SYSTEM washer_detector
  (* Version 1.0, 2024-11-25, obotnar *)
  APPLICATION washer_detectorApp
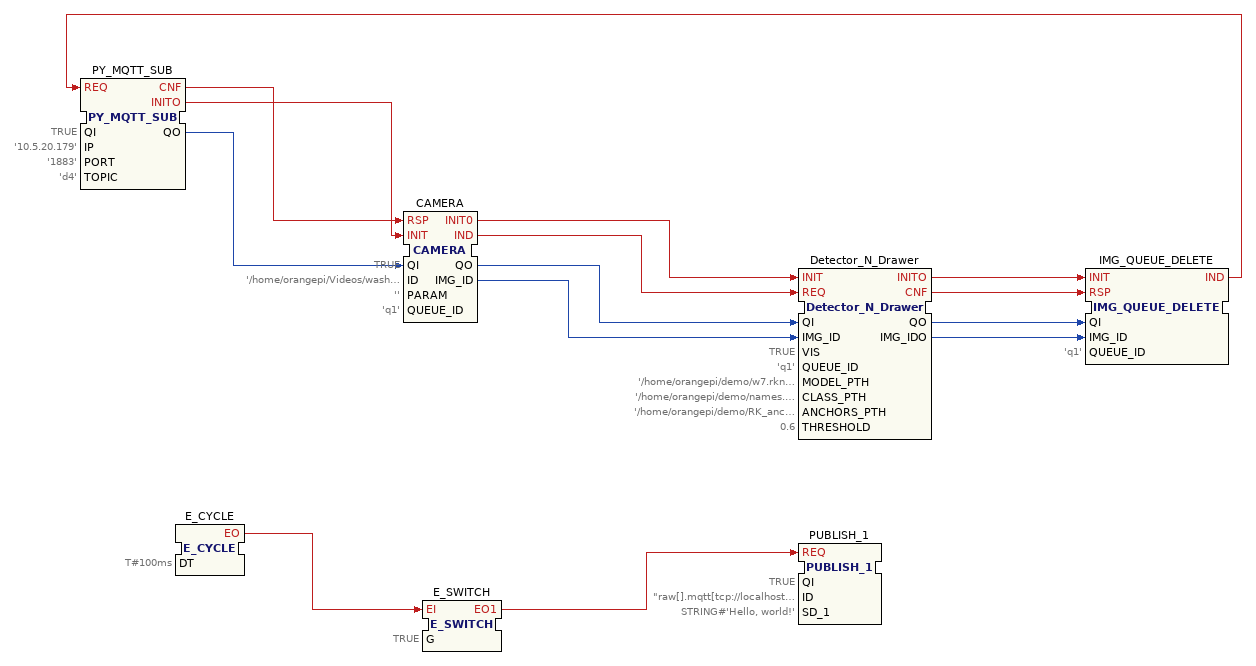
    FBS
      CAMERA : CAMERA(QI := TRUE, ID := '/home/orangepi/Videos/washer.webm', PARAM := '', QUEUE_ID := 'q1');
      IMG_QUEUE_DELETE : IMG_QUEUE_DELETE(QUEUE_ID := 'q1');
      Detector_N_Drawer : Detector_N_Drawer(VIS := TRUE, QUEUE_ID := 'q1', MODEL_PTH := '/home/orangepi/demo/w7.rknn', CLASS_PTH := '/home/orangepi/demo/names.txt', ANCHORS_PTH := '/home/orangepi/demo/RK_anchors.txt', THRESHOLD := 0.6);
      PY_MQTT_SUB : PY_MQTT_SUB(QI := TRUE, IP := '10.5.20.179', PORT := '1883', TOPIC := 'd4');
      E_SWITCH : E_SWITCH(G := TRUE);
      PUBLISH_1 : PUBLISH_1(QI := TRUE, ID := "raw[].mqtt[tcp://localhost:1883, forte, d4]", SD_1 := STRING#'Hello, world!');
      E_CYCLE : E_CYCLE(DT := T#100ms);
    END_FBS
    EVENT_CONNECTIONS
      CAMERA.INIT0 TO Detector_N_Drawer.INIT;
      CAMERA.IND TO Detector_N_Drawer.REQ;
      Detector_N_Drawer.INITO TO IMG_QUEUE_DELETE.INIT;
      Detector_N_Drawer.CNF TO IMG_QUEUE_DELETE.RSP;
      PY_MQTT_SUB.CNF TO CAMERA.RSP;
      PY_MQTT_SUB.INITO TO CAMERA.INIT;
      IMG_QUEUE_DELETE.IND TO PY_MQTT_SUB.REQ;
      E_SWITCH.EO1 TO PUBLISH_1.REQ;
      E_CYCLE.EO TO E_SWITCH.EI;
    END_CONNECTIONS
    DATA_CONNECTIONS
      Detector_N_Drawer.QO TO IMG_QUEUE_DELETE.QI;
      Detector_N_Drawer.IMG_IDO TO IMG_QUEUE_DELETE.IMG_ID;
      CAMERA.QO TO Detector_N_Drawer.QI;
      CAMERA.IMG_ID TO Detector_N_Drawer.IMG_ID;
      PY_MQTT_SUB.QO TO CAMERA.QI;
    END_CONNECTIONS
  END_APPLICATION
  DEVICE FORTE_PC : FORTE_PC(MGR_ID := "10.5.20.198:62499" (* Device manager socket ID *))
    {SET_ATTRIBUTE(Profile, HOLOBLOC)}
    RESOURCE EMB_RES : EMB_RES
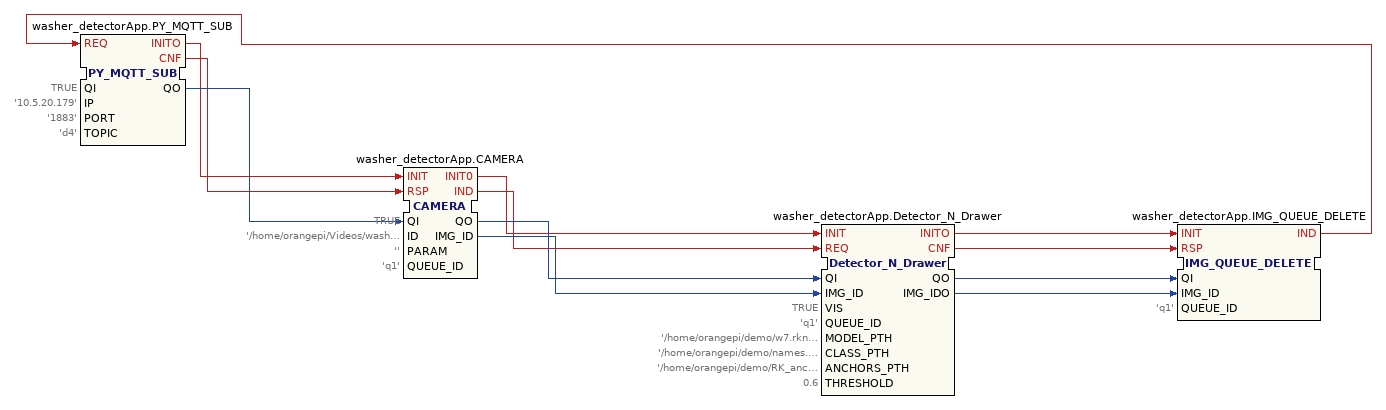
      FBS
        washer_detectorApp.PY_MQTT_SUB : PY_MQTT_SUB(QI := TRUE, IP := '10.5.20.179', PORT := '1883', TOPIC := 'd4');
        washer_detectorApp.CAMERA : CAMERA(QI := TRUE, ID := '/home/orangepi/Videos/washer.webm', PARAM := '', QUEUE_ID := 'q1');
        washer_detectorApp.Detector_N_Drawer : Detector_N_Drawer(VIS := TRUE, QUEUE_ID := 'q1', MODEL_PTH := '/home/orangepi/demo/w7.rknn', CLASS_PTH := '/home/orangepi/demo/names.txt', ANCHORS_PTH := '/home/orangepi/demo/RK_anchors.txt', THRESHOLD := 0.6);
        washer_detectorApp.IMG_QUEUE_DELETE : IMG_QUEUE_DELETE(QUEUE_ID := 'q1');
      END_FBS
      EVENT_CONNECTIONS
        washer_detectorApp.PY_MQTT_SUB.INITO TO washer_detectorApp.CAMERA.INIT;
        washer_detectorApp.PY_MQTT_SUB.CNF TO washer_detectorApp.CAMERA.RSP;
        washer_detectorApp.CAMERA.INIT0 TO washer_detectorApp.Detector_N_Drawer.INIT;
        washer_detectorApp.CAMERA.IND TO washer_detectorApp.Detector_N_Drawer.REQ;
        washer_detectorApp.Detector_N_Drawer.INITO TO washer_detectorApp.IMG_QUEUE_DELETE.INIT;
        washer_detectorApp.Detector_N_Drawer.CNF TO washer_detectorApp.IMG_QUEUE_DELETE.RSP;
        washer_detectorApp.IMG_QUEUE_DELETE.IND TO washer_detectorApp.PY_MQTT_SUB.REQ;
      END_CONNECTIONS
      DATA_CONNECTIONS
        washer_detectorApp.PY_MQTT_SUB.QO TO washer_detectorApp.CAMERA.QI;
        washer_detectorApp.CAMERA.QO TO washer_detectorApp.Detector_N_Drawer.QI;
        washer_detectorApp.CAMERA.IMG_ID TO washer_detectorApp.Detector_N_Drawer.IMG_ID;
        washer_detectorApp.Detector_N_Drawer.QO TO washer_detectorApp.IMG_QUEUE_DELETE.QI;
        washer_detectorApp.Detector_N_Drawer.IMG_IDO TO washer_detectorApp.IMG_QUEUE_DELETE.IMG_ID;
      END_CONNECTIONS
    END_RESOURCE
  END_DEVICE
  DEVICE FORTE_PC_1 : FORTE_PC(MGR_ID := "localhost:61499" (* Device manager socket ID *))
    {SET_ATTRIBUTE(Profile, HOLOBLOC)}
    RESOURCE EMB_RES : EMB_RES
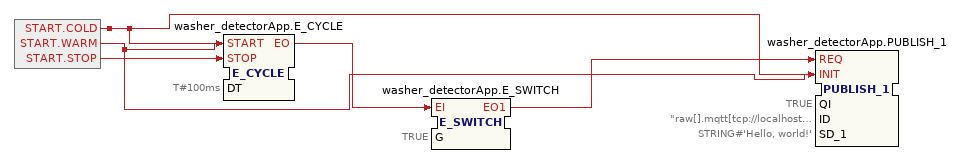
      FBS
        washer_detectorApp.PUBLISH_1 : PUBLISH_1(QI := TRUE, ID := "raw[].mqtt[tcp://localhost:1883, forte, d4]", SD_1 := STRING#'Hello, world!');
        washer_detectorApp.E_SWITCH : E_SWITCH(G := TRUE);
        washer_detectorApp.E_CYCLE : E_CYCLE(DT := T#100ms);
      END_FBS
      EVENT_CONNECTIONS
        washer_detectorApp.E_SWITCH.EO1 TO washer_detectorApp.PUBLISH_1.REQ;
        washer_detectorApp.E_CYCLE.EO TO washer_detectorApp.E_SWITCH.EI;
        START.COLD TO washer_detectorApp.E_CYCLE.START;
        START.WARM TO washer_detectorApp.E_CYCLE.START;
        START.STOP TO washer_detectorApp.E_CYCLE.STOP;
        START.COLD TO washer_detectorApp.PUBLISH_1.INIT;
        START.WARM TO washer_detectorApp.PUBLISH_1.INIT;
      END_CONNECTIONS
    END_RESOURCE
  END_DEVICE
  MAPPINGS
    washer_detectorApp.CAMERA ON FORTE_PC.EMB_RES;
    washer_detectorApp.IMG_QUEUE_DELETE ON FORTE_PC.EMB_RES;
    washer_detectorApp.Detector_N_Drawer ON FORTE_PC.EMB_RES;
    washer_detectorApp.PY_MQTT_SUB ON FORTE_PC.EMB_RES;
    washer_detectorApp.PUBLISH_1 ON FORTE_PC_1.EMB_RES;
    washer_detectorApp.E_SWITCH ON FORTE_PC_1.EMB_RES;
    washer_detectorApp.E_CYCLE ON FORTE_PC_1.EMB_RES;
  END_MAPPINGS
  SEGMENTS
    Ethernet : Ethernet;
  END_SEGMENTS
  LINKS
    FORTE_PC => Ethernet;
    FORTE_PC_1 => Ethernet;
  END_LINKS
END_SYSTEM
